# EPICS autosave request: ARAmpApp/Db/aramp_settings_75A400.req
# This file specifies which PVs of the corresponding database should be saved.

# Gain
$(P)$(R)Gain-SP

# Lock Gain dB with Gain in steps
$(P)$(R)GainAuto-Sel

# Enable
$(P)$(R)Enbl-Sel
